// TIA Portal V17 export
// export: Created 2025-03-05T08:00:13.2109361Z, ExportSetting WithDefaults, DisplayName Totally Integrated Automation Portal, DisplayVersion V17 Update 8, DisplayName TIA Portal Openness, DisplayVersion V17 Update 8, DisplayName TIA Portal Version Control Interface, DisplayVersion V17, DisplayName SINAMICS Startdrive Advanced, DisplayVersion V17 SP2, DisplayName SINAMICS Startdrive G110M, G120, G120C, G120D, G120P, G115D, DisplayVersion V17 SP2, DisplayName SINAMICS Startdrive G130, G150, S120, S150, SINAMICS MV, S210, DisplayVersion V17 SP2, DisplayName STEP 7 Professional, DisplayVersion V17 Update 8, DisplayName SINUMERIK ONE STEP 7 Toolbox, DisplayVersion V17 Update 12, DisplayName SINUMERIK 840D sl STEP 7 Toolbox, DisplayVersion V17 Update 12, DisplayName STEP 7 Safety, DisplayVersion V17 Update 6, DisplayName WinCC Advanced, DisplayVersion V17 Update 8
FUNCTION "FC2108_MACHINE_CONTROL_ON" : Void   // FC2108, LAD
{ S7_Optimized_Access := 'FALSE' }
AUTHOR : ETXETAR
VERSION : 1.0
// stored: AutoNumber false, IsIECCheckEnabled false, SetENOAutomatically false, UDAEnableTagReadback false
   VAR_TEMP
      O_BYTE_0 : Struct   // OPTIONS BYTE 0
         GM_COOLANT_PUMP_OFF_DELAY : Bool;   // GM COOLANT PUMP POWER OFF DELAY OPTION
      END_STRUCT;
   END_VAR
   VAR CONSTANT
      FC_NUMBER : DInt := 2108;   // FC NUMBER
   END_VAR
   VAR_TEMP   // added for the SCL form of the ladder/FBD networks
      _w1 : Bool;
   END_VAR
BEGIN

REGION Network 1: OPTIONS
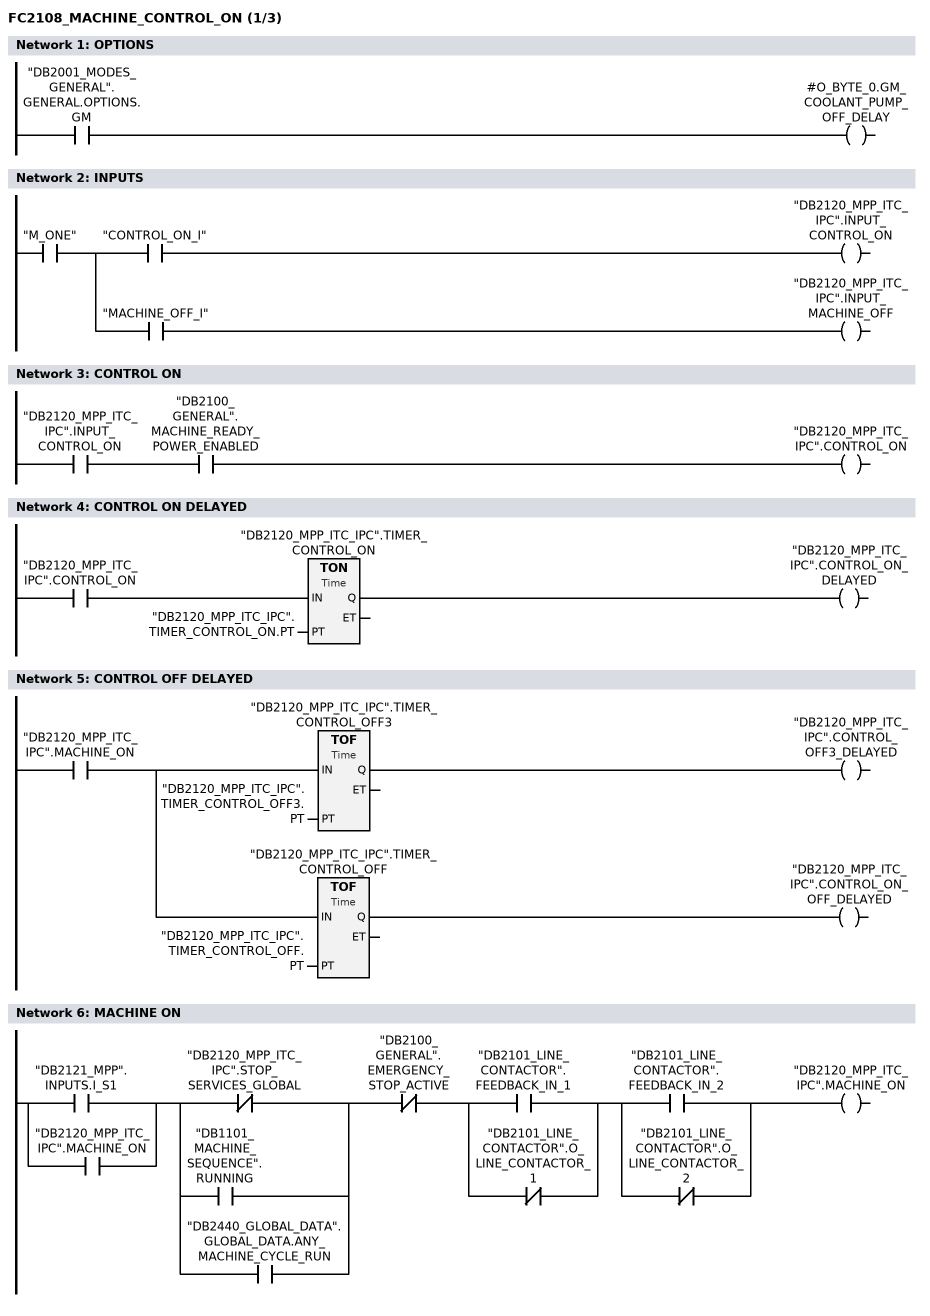
   RUNG wire#powerrail
      Contact( "DB2001_MODES_GENERAL".GENERAL.OPTIONS.GM )
      Coil( #O_BYTE_0.GM_COOLANT_PUMP_OFF_DELAY )
   END_RUNG
   // the same network as SCL:
   #O_BYTE_0.GM_COOLANT_PUMP_OFF_DELAY := "DB2001_MODES_GENERAL".GENERAL.OPTIONS.GM;
END_REGION

REGION Network 2: INPUTS
   RUNG wire#powerrail
      Contact( "M_ONE" )
      wire#w1
      Contact( "CONTROL_ON_I" )
      Coil( "DB2120_MPP_ITC_IPC".INPUT_CONTROL_ON )
   END_RUNG
   RUNG wire#w1
      Contact( "MACHINE_OFF_I" )
      Coil( "DB2120_MPP_ITC_IPC".INPUT_MACHINE_OFF )
   END_RUNG
   // the same network as SCL:
   "DB2120_MPP_ITC_IPC".INPUT_CONTROL_ON := "M_ONE" AND "CONTROL_ON_I";
   "DB2120_MPP_ITC_IPC".INPUT_MACHINE_OFF := "M_ONE" AND "MACHINE_OFF_I";
END_REGION

REGION Network 3: CONTROL ON
   RUNG wire#powerrail
      Contact( "DB2120_MPP_ITC_IPC".INPUT_CONTROL_ON )
      Contact( "DB2100_GENERAL".MACHINE_READY_POWER_ENABLED )
      Coil( "DB2120_MPP_ITC_IPC".CONTROL_ON )
   END_RUNG
   // the same network as SCL:
   "DB2120_MPP_ITC_IPC".CONTROL_ON := "DB2120_MPP_ITC_IPC".INPUT_CONTROL_ON AND "DB2100_GENERAL".MACHINE_READY_POWER_ENABLED;
END_REGION

REGION Network 4: CONTROL ON DELAYED
   RUNG wire#powerrail
      Contact( "DB2120_MPP_ITC_IPC".CONTROL_ON )
      { S7_Templates := "time_type := Time" } "DB2120_MPP_ITC_IPC".TIMER_CONTROL_ON.TON(pt := "DB2120_MPP_ITC_IPC".TIMER_CONTROL_ON.PT, et =>)
      Coil( "DB2120_MPP_ITC_IPC".CONTROL_ON_DELAYED )
   END_RUNG
   // the same network as SCL:
   "DB2120_MPP_ITC_IPC".TIMER_CONTROL_ON.TON(IN := "DB2120_MPP_ITC_IPC".CONTROL_ON,
                           PT := "DB2120_MPP_ITC_IPC".TIMER_CONTROL_ON.PT);
   "DB2120_MPP_ITC_IPC".CONTROL_ON_DELAYED := "DB2120_MPP_ITC_IPC".TIMER_CONTROL_ON.Q;
END_REGION

REGION Network 5: CONTROL OFF DELAYED
   RUNG wire#powerrail
      Contact( "DB2120_MPP_ITC_IPC".MACHINE_ON )
      wire#w1
      { S7_Templates := "time_type := Time" } "DB2120_MPP_ITC_IPC".TIMER_CONTROL_OFF3.TOF(pt := "DB2120_MPP_ITC_IPC".TIMER_CONTROL_OFF3.PT, et =>)
      Coil( "DB2120_MPP_ITC_IPC".CONTROL_OFF3_DELAYED )
   END_RUNG
   RUNG wire#w1
      { S7_Templates := "time_type := Time" } "DB2120_MPP_ITC_IPC".TIMER_CONTROL_OFF.TOF(pt := "DB2120_MPP_ITC_IPC".TIMER_CONTROL_OFF.PT, et =>)
      Coil( "DB2120_MPP_ITC_IPC".CONTROL_ON_OFF_DELAYED )
   END_RUNG
   // the same network as SCL:
   "DB2120_MPP_ITC_IPC".TIMER_CONTROL_OFF3.TOF(IN := "DB2120_MPP_ITC_IPC".MACHINE_ON,
                           PT := "DB2120_MPP_ITC_IPC".TIMER_CONTROL_OFF3.PT);
   "DB2120_MPP_ITC_IPC".CONTROL_OFF3_DELAYED := "DB2120_MPP_ITC_IPC".TIMER_CONTROL_OFF3.Q;
   "DB2120_MPP_ITC_IPC".TIMER_CONTROL_OFF.TOF(IN := "DB2120_MPP_ITC_IPC".MACHINE_ON,
                           PT := "DB2120_MPP_ITC_IPC".TIMER_CONTROL_OFF.PT);
   "DB2120_MPP_ITC_IPC".CONTROL_ON_OFF_DELAYED := "DB2120_MPP_ITC_IPC".TIMER_CONTROL_OFF.Q;
END_REGION

REGION Network 6: MACHINE ON
   RUNG wire#powerrail
      Contact( "DB2121_MPP".INPUTS.I_S1 )
      wire#w1
      I_Contact( "DB2120_MPP_ITC_IPC".STOP_SERVICES_GLOBAL )
      wire#w2
      I_Contact( "DB2100_GENERAL".EMERGENCY_STOP_ACTIVE )
      wire#w3
      Contact( "DB2101_LINE_CONTACTOR".FEEDBACK_IN_1 )
      wire#w4
      Contact( "DB2101_LINE_CONTACTOR".FEEDBACK_IN_2 )
      wire#w5
      Coil( "DB2120_MPP_ITC_IPC".MACHINE_ON )
   END_RUNG
   RUNG wire#powerrail
      Contact( "DB2120_MPP_ITC_IPC".MACHINE_ON )
   END_RUNG wire#w1
   RUNG wire#w1
      Contact( "DB1101_MACHINE_SEQUENCE".RUNNING )
   END_RUNG wire#w2
   RUNG wire#w1
      Contact( "DB2440_GLOBAL_DATA".GLOBAL_DATA.ANY_MACHINE_CYCLE_RUN )
   END_RUNG wire#w2
   RUNG wire#w3
      I_Contact( "DB2101_LINE_CONTACTOR".O_LINE_CONTACTOR_1 )
   END_RUNG wire#w4
   RUNG wire#w4
      I_Contact( "DB2101_LINE_CONTACTOR".O_LINE_CONTACTOR_2 )
   END_RUNG wire#w5
   // the same network as SCL:
   "DB2120_MPP_ITC_IPC".MACHINE_ON := ("DB2121_MPP".INPUTS.I_S1 OR "DB2120_MPP_ITC_IPC".MACHINE_ON) AND (NOT "DB2120_MPP_ITC_IPC".STOP_SERVICES_GLOBAL OR "DB1101_MACHINE_SEQUENCE".RUNNING OR "DB2440_GLOBAL_DATA".GLOBAL_DATA.ANY_MACHINE_CYCLE_RUN) AND NOT "DB2100_GENERAL".EMERGENCY_STOP_ACTIVE AND ("DB2101_LINE_CONTACTOR".FEEDBACK_IN_1 OR NOT "DB2101_LINE_CONTACTOR".O_LINE_CONTACTOR_1) AND ("DB2101_LINE_CONTACTOR".FEEDBACK_IN_2 OR NOT "DB2101_LINE_CONTACTOR".O_LINE_CONTACTOR_2);
END_REGION

REGION Network 7: MACHINE ON DELAYED
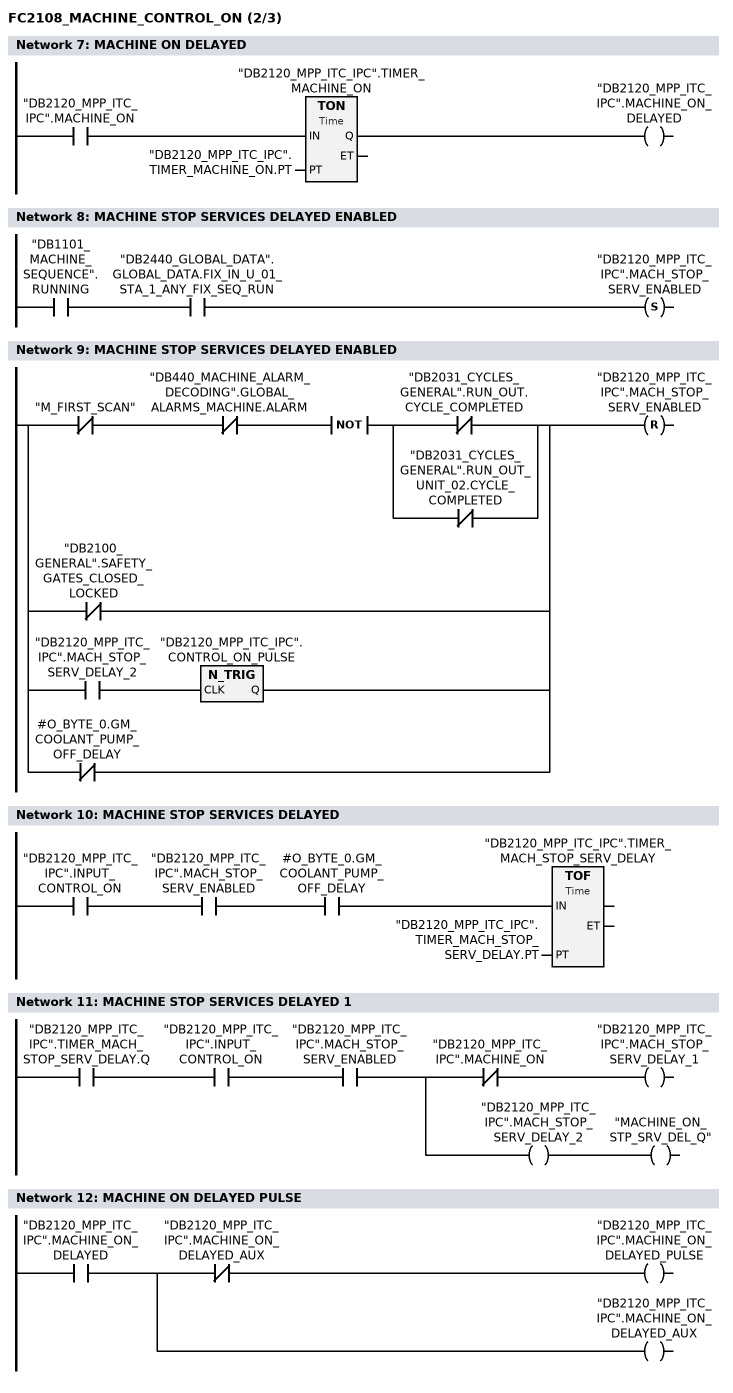
   RUNG wire#powerrail
      Contact( "DB2120_MPP_ITC_IPC".MACHINE_ON )
      { S7_Templates := "time_type := Time" } "DB2120_MPP_ITC_IPC".TIMER_MACHINE_ON.TON(pt := "DB2120_MPP_ITC_IPC".TIMER_MACHINE_ON.PT, et =>)
      Coil( "DB2120_MPP_ITC_IPC".MACHINE_ON_DELAYED )
   END_RUNG
   // the same network as SCL:
   "DB2120_MPP_ITC_IPC".TIMER_MACHINE_ON.TON(IN := "DB2120_MPP_ITC_IPC".MACHINE_ON,
                           PT := "DB2120_MPP_ITC_IPC".TIMER_MACHINE_ON.PT);
   "DB2120_MPP_ITC_IPC".MACHINE_ON_DELAYED := "DB2120_MPP_ITC_IPC".TIMER_MACHINE_ON.Q;
END_REGION

REGION Network 8: MACHINE STOP SERVICES DELAYED ENABLED
   RUNG wire#powerrail
      Contact( "DB1101_MACHINE_SEQUENCE".RUNNING )
      Contact( "DB2440_GLOBAL_DATA".GLOBAL_DATA.FIX_IN_U_01_STA_1_ANY_FIX_SEQ_RUN )
      S_Coil( "DB2120_MPP_ITC_IPC".MACH_STOP_SERV_ENABLED )
   END_RUNG
   // the same network as SCL:
   IF "DB1101_MACHINE_SEQUENCE".RUNNING AND "DB2440_GLOBAL_DATA".GLOBAL_DATA.FIX_IN_U_01_STA_1_ANY_FIX_SEQ_RUN THEN
       "DB2120_MPP_ITC_IPC".MACH_STOP_SERV_ENABLED := TRUE;
   END_IF;
END_REGION

REGION Network 9: MACHINE STOP SERVICES DELAYED ENABLED
   RUNG wire#powerrail
      I_Contact( "M_FIRST_SCAN" )
      I_Contact( "DB440_MACHINE_ALARM_DECODING".GLOBAL_ALARMS_MACHINE.ALARM )
      Not()
      wire#w1
      I_Contact( "DB2031_CYCLES_GENERAL".RUN_OUT.CYCLE_COMPLETED )
      wire#w2
      R_Coil( "DB2120_MPP_ITC_IPC".MACH_STOP_SERV_ENABLED )
   END_RUNG
   RUNG wire#w1
      I_Contact( "DB2031_CYCLES_GENERAL".RUN_OUT_UNIT_02.CYCLE_COMPLETED )
   END_RUNG wire#w2
   RUNG wire#powerrail
      I_Contact( "DB2100_GENERAL".SAFETY_GATES_CLOSED_LOCKED )
   END_RUNG wire#w2
   RUNG wire#powerrail
      Contact( "DB2120_MPP_ITC_IPC".MACH_STOP_SERV_DELAY_2 )
      N_Trig( "DB2120_MPP_ITC_IPC".CONTROL_ON_PULSE )
   END_RUNG wire#w2
   RUNG wire#powerrail
      I_Contact( #O_BYTE_0.GM_COOLANT_PUMP_OFF_DELAY )
   END_RUNG wire#w2
   // the same network as SCL:
   #_w1 := NOT "DB2120_MPP_ITC_IPC".MACH_STOP_SERV_DELAY_2 AND "DB2120_MPP_ITC_IPC".CONTROL_ON_PULSE;   // falling edge
   "DB2120_MPP_ITC_IPC".CONTROL_ON_PULSE := "DB2120_MPP_ITC_IPC".MACH_STOP_SERV_DELAY_2;
   IF (NOT (NOT "M_FIRST_SCAN" AND NOT "DB440_MACHINE_ALARM_DECODING".GLOBAL_ALARMS_MACHINE.ALARM) AND (NOT "DB2031_CYCLES_GENERAL".RUN_OUT.CYCLE_COMPLETED OR NOT "DB2031_CYCLES_GENERAL".RUN_OUT_UNIT_02.CYCLE_COMPLETED)) OR NOT "DB2100_GENERAL".SAFETY_GATES_CLOSED_LOCKED OR #_w1 OR NOT #O_BYTE_0.GM_COOLANT_PUMP_OFF_DELAY THEN
       "DB2120_MPP_ITC_IPC".MACH_STOP_SERV_ENABLED := FALSE;
   END_IF;
END_REGION

REGION Network 10: MACHINE STOP SERVICES DELAYED
   RUNG wire#powerrail
      Contact( "DB2120_MPP_ITC_IPC".INPUT_CONTROL_ON )
      Contact( "DB2120_MPP_ITC_IPC".MACH_STOP_SERV_ENABLED )
      Contact( #O_BYTE_0.GM_COOLANT_PUMP_OFF_DELAY )
      { S7_Templates := "time_type := Time" } "DB2120_MPP_ITC_IPC".TIMER_MACH_STOP_SERV_DELAY.TOF(pt := "DB2120_MPP_ITC_IPC".TIMER_MACH_STOP_SERV_DELAY.PT, et =>)
   END_RUNG
   // the same network as SCL:
   "DB2120_MPP_ITC_IPC".TIMER_MACH_STOP_SERV_DELAY.TOF(IN := "DB2120_MPP_ITC_IPC".INPUT_CONTROL_ON AND "DB2120_MPP_ITC_IPC".MACH_STOP_SERV_ENABLED AND #O_BYTE_0.GM_COOLANT_PUMP_OFF_DELAY,
                           PT := "DB2120_MPP_ITC_IPC".TIMER_MACH_STOP_SERV_DELAY.PT);
END_REGION

REGION Network 11: MACHINE STOP SERVICES DELAYED 1
   RUNG wire#powerrail
      Contact( "DB2120_MPP_ITC_IPC".TIMER_MACH_STOP_SERV_DELAY.Q )
      Contact( "DB2120_MPP_ITC_IPC".INPUT_CONTROL_ON )
      Contact( "DB2120_MPP_ITC_IPC".MACH_STOP_SERV_ENABLED )
      wire#w1
      I_Contact( "DB2120_MPP_ITC_IPC".MACHINE_ON )
      Coil( "DB2120_MPP_ITC_IPC".MACH_STOP_SERV_DELAY_1 )
   END_RUNG
   RUNG wire#w1
      Coil( "DB2120_MPP_ITC_IPC".MACH_STOP_SERV_DELAY_2 )
      Coil( "MACHINE_ON_STP_SRV_DEL_Q" )
   END_RUNG
   // the same network as SCL:
   #_w1 := "DB2120_MPP_ITC_IPC".TIMER_MACH_STOP_SERV_DELAY.Q AND "DB2120_MPP_ITC_IPC".INPUT_CONTROL_ON AND "DB2120_MPP_ITC_IPC".MACH_STOP_SERV_ENABLED;
   "DB2120_MPP_ITC_IPC".MACH_STOP_SERV_DELAY_1 := #_w1 AND NOT "DB2120_MPP_ITC_IPC".MACHINE_ON;
   "DB2120_MPP_ITC_IPC".MACH_STOP_SERV_DELAY_2 := #_w1;
   "MACHINE_ON_STP_SRV_DEL_Q" := #_w1;
END_REGION

REGION Network 12: MACHINE ON DELAYED PULSE
   RUNG wire#powerrail
      Contact( "DB2120_MPP_ITC_IPC".MACHINE_ON_DELAYED )
      wire#w1
      I_Contact( "DB2120_MPP_ITC_IPC".MACHINE_ON_DELAYED_AUX )
      Coil( "DB2120_MPP_ITC_IPC".MACHINE_ON_DELAYED_PULSE )
   END_RUNG
   RUNG wire#w1
      Coil( "DB2120_MPP_ITC_IPC".MACHINE_ON_DELAYED_AUX )
   END_RUNG
   // the same network as SCL:
   "DB2120_MPP_ITC_IPC".MACHINE_ON_DELAYED_PULSE := "DB2120_MPP_ITC_IPC".MACHINE_ON_DELAYED AND NOT "DB2120_MPP_ITC_IPC".MACHINE_ON_DELAYED_AUX;
   "DB2120_MPP_ITC_IPC".MACHINE_ON_DELAYED_AUX := "DB2120_MPP_ITC_IPC".MACHINE_ON_DELAYED;
END_REGION

REGION Network 13: MACHINE OFF DELAYED
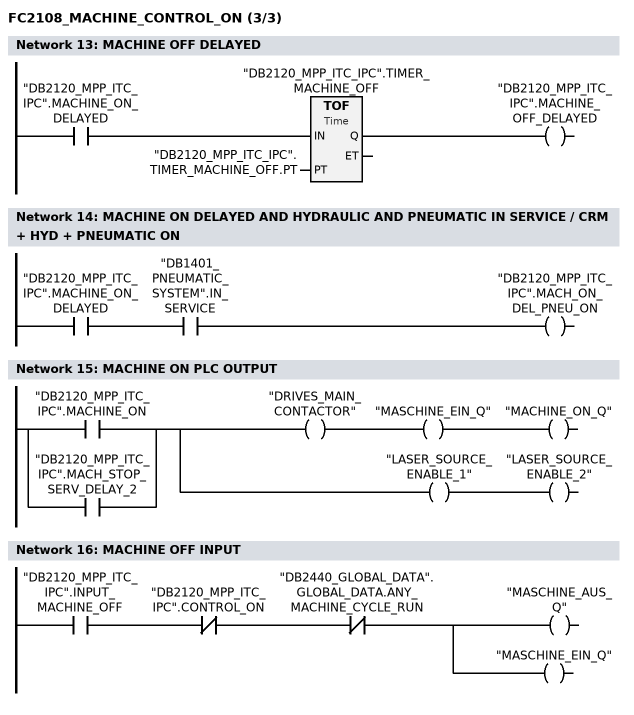
   RUNG wire#powerrail
      Contact( "DB2120_MPP_ITC_IPC".MACHINE_ON_DELAYED )
      { S7_Templates := "time_type := Time" } "DB2120_MPP_ITC_IPC".TIMER_MACHINE_OFF.TOF(pt := "DB2120_MPP_ITC_IPC".TIMER_MACHINE_OFF.PT, et =>)
      Coil( "DB2120_MPP_ITC_IPC".MACHINE_OFF_DELAYED )
   END_RUNG
   // the same network as SCL:
   "DB2120_MPP_ITC_IPC".TIMER_MACHINE_OFF.TOF(IN := "DB2120_MPP_ITC_IPC".MACHINE_ON_DELAYED,
                           PT := "DB2120_MPP_ITC_IPC".TIMER_MACHINE_OFF.PT);
   "DB2120_MPP_ITC_IPC".MACHINE_OFF_DELAYED := "DB2120_MPP_ITC_IPC".TIMER_MACHINE_OFF.Q;
END_REGION

REGION Network 14: MACHINE ON DELAYED AND HYDRAULIC AND PNEUMATIC IN SERVICE / CRM + HYD + PNEUMATIC ON
   RUNG wire#powerrail
      Contact( "DB2120_MPP_ITC_IPC".MACHINE_ON_DELAYED )
      Contact( "DB1401_PNEUMATIC_SYSTEM".IN_SERVICE )
      Coil( "DB2120_MPP_ITC_IPC".MACH_ON_DEL_PNEU_ON )
   END_RUNG
   // the same network as SCL:
   "DB2120_MPP_ITC_IPC".MACH_ON_DEL_PNEU_ON := "DB2120_MPP_ITC_IPC".MACHINE_ON_DELAYED AND "DB1401_PNEUMATIC_SYSTEM".IN_SERVICE;
END_REGION

REGION Network 15: MACHINE ON PLC OUTPUT
   RUNG wire#powerrail
      Contact( "DB2120_MPP_ITC_IPC".MACHINE_ON )
      wire#w1
      Coil( "DRIVES_MAIN_CONTACTOR" )
      Coil( "MASCHINE_EIN_Q" )
      Coil( "MACHINE_ON_Q" )
   END_RUNG
   RUNG wire#powerrail
      Contact( "DB2120_MPP_ITC_IPC".MACH_STOP_SERV_DELAY_2 )
   END_RUNG wire#w1
   RUNG wire#w1
      Coil( "LASER_SOURCE_ENABLE_1" )
      Coil( "LASER_SOURCE_ENABLE_2" )
   END_RUNG
   // the same network as SCL:
   "DRIVES_MAIN_CONTACTOR" := "DB2120_MPP_ITC_IPC".MACHINE_ON OR "DB2120_MPP_ITC_IPC".MACH_STOP_SERV_DELAY_2;
   "MASCHINE_EIN_Q" := "DRIVES_MAIN_CONTACTOR";
   "MACHINE_ON_Q" := "DRIVES_MAIN_CONTACTOR";
   "LASER_SOURCE_ENABLE_1" := "DRIVES_MAIN_CONTACTOR";
   "LASER_SOURCE_ENABLE_2" := "DRIVES_MAIN_CONTACTOR";
END_REGION

REGION Network 16: MACHINE OFF INPUT
   RUNG wire#powerrail
      Contact( "DB2120_MPP_ITC_IPC".INPUT_MACHINE_OFF )
      I_Contact( "DB2120_MPP_ITC_IPC".CONTROL_ON )
      I_Contact( "DB2440_GLOBAL_DATA".GLOBAL_DATA.ANY_MACHINE_CYCLE_RUN )
      wire#w1
      Coil( "MASCHINE_AUS_Q" )
   END_RUNG
   RUNG wire#w1
      Coil( "MASCHINE_EIN_Q" )
   END_RUNG
   // the same network as SCL:
   "MASCHINE_AUS_Q" := "DB2120_MPP_ITC_IPC".INPUT_MACHINE_OFF AND NOT "DB2120_MPP_ITC_IPC".CONTROL_ON AND NOT "DB2440_GLOBAL_DATA".GLOBAL_DATA.ANY_MACHINE_CYCLE_RUN;
   "MASCHINE_EIN_Q" := "MASCHINE_AUS_Q";
END_REGION
END_FUNCTION
